TYPE ST_RobotRegionMove_Info :
STRUCT
	Get				: BOOL;
	UseA			: BOOL;
	UseB			: BOOL;
	A_Position		: LREAL;
	B_Position		: LREAL;
END_STRUCT
END_TYPE

(* stored: Version 1.1.0.1, ProductVersion 3.1.4024.13
   DUT ST_RobotRegionMove_Info: Id {109977ff-f048-4d74-9b7a-27ae1e51120f} *)
